# EPICS autosave request: iocBoot/ioc13HG100/auto_settings.req
file "HG-100_settings.req",      P=$(P), R=HG100:
#file "pid_control_settings.req"  P=$(P), PID=PID1
